(* Logix 5000 project; controller Modbus_TCP_Client_Example vendor 1 type 14 code 154 rev 32.15; software revision 32.05; part 7 of 10 *)

ADD_ON_INSTRUCTION AMP_SCL_Command_Execute   (* revision 1.0 *)
// Applied Motion - SCL Command Execute AOI
// Help:
// The SCL Command Execute AOI executes selected SCL commands (as listed under “Available SCL Commands” in the Host Command Reference).
VAR_IN_OUT
   Input : DINT[14]; {required}   // Drive Input Assembly
   Output : DINT[16]; {required}   // Drive Output Assembly
        [0]   // Command Word
        [10]   // Data/Register 1
        [11]   // Data/Register 2
        [1]   // Jog Speed (0.25 rev/min)
        [2]   // Jog Acceleration (10 rev/s/s)
        [3]   // Jog Deceleration (10 rev/s/s)
        [4]   // Point-to-Point Velocity (0.25 rev/min)
        [5]   // Point-to-Point Acceleration (10 rev/s/s)
        [6]   // Point-to-Point Deceleration (10 rev/s/s)
        [7]   // Point-to-Point Distance (Motor steps)
        [9]   // (2x ASCII Letters in 16 lower word)
END_VAR
VAR_INPUT
   RPI : DINT := 100; {visible}   // Drive Connection Request Packet Interval (milliseconds)
   Execute : BOOL; {required}   // Execute the SCL command
   SCL_Command : INT; {required}   // SCL Command Characters (always 2)
   Reg1 : DINT; {required}   // Data / SCL Register 1
   Reg2 : DINT; {required}   // Data / SCL Register 2
END_VAR
VAR_OUTPUT
   Sent : BOOL; {access Read Only, visible}   // Command has been sent to drive
   In_Progress : BOOL; {access Read Only, visible}   // In progress = sending command
   Done : BOOL; {access Read Only, visible}   // Command sent
   Error : BOOL; {access Read Only, visible}   // Command failed to be sent
   State : DINT := 10; {access Read Only}   // Internal state of progress
END_VAR
VAR
   Loc_StatusCode : AMP_Status_Word;
   Loc_CommandOff_Timer : TIMER;   // Timer to make sure command value was 0 before sending a new command
   Loc_CommandOn_Timer : TIMER;   // Timer to make sure command value is set long enough to be sent to drive
   Loc_Input_Assembly : AMP_Input_Assembly_v2; {access None}
   Loc_Start_ONS : BOOL; {access None}
END_VAR

ROUTINE Logic   (* ladder *)
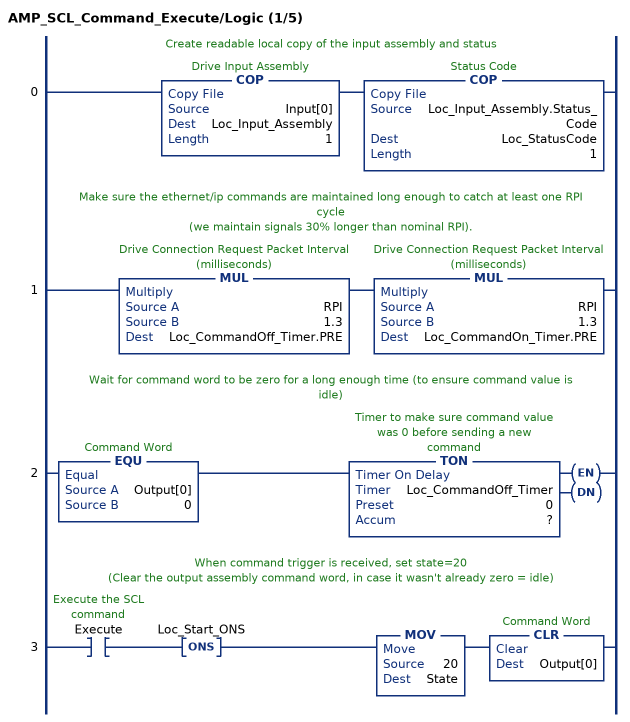
   // Create readable local copy of the input assembly and status
   0: COP(Input[0],Loc_Input_Assembly,1)COP(Loc_Input_Assembly.Status_Code,Loc_StatusCode,1);
   // Make sure the ethernet/ip commands are maintained long enough to catch at least one RPI cycle
   // (we maintain signals 30% longer than nominal RPI).
   1: MUL(RPI,1.3,Loc_CommandOff_Timer.PRE)MUL(RPI,1.3,Loc_CommandOn_Timer.PRE);
   // Wait for command word to be zero for a long enough time (to ensure command value is idle)
   2: EQU(Output[0],0)TON(Loc_CommandOff_Timer,?,?);
   // When command trigger is received, set state=20
   // (Clear the output assembly command word, in case it wasn't already zero = idle)
   3: XIC(Execute)ONS(Loc_Start_ONS)MOV(20,State)CLR(Output[0]);
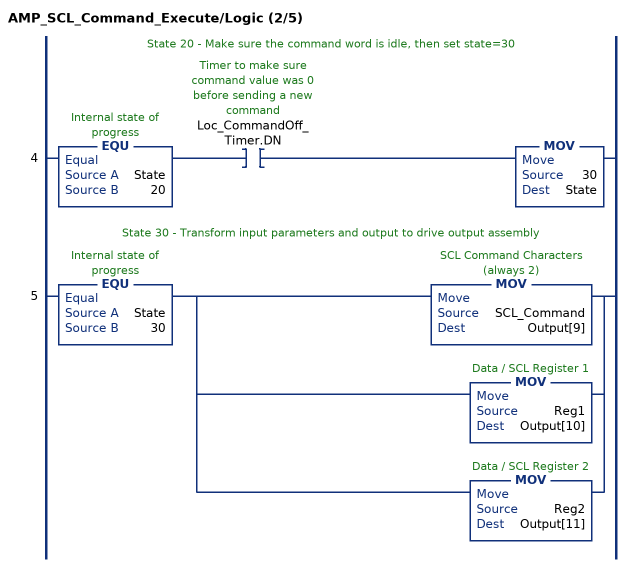
   // State 20 - Make sure the command word is idle, then set state=30
   4: EQU(State,20)XIC(Loc_CommandOff_Timer.DN)MOV(30,State);
   // State 30 - Transform input parameters and output to drive output assembly
   5: EQU(State,30)[MOV(SCL_Command,Output[9]) ,MOV(Reg1,Output[10]) ,MOV(Reg2,Output[11]) ];
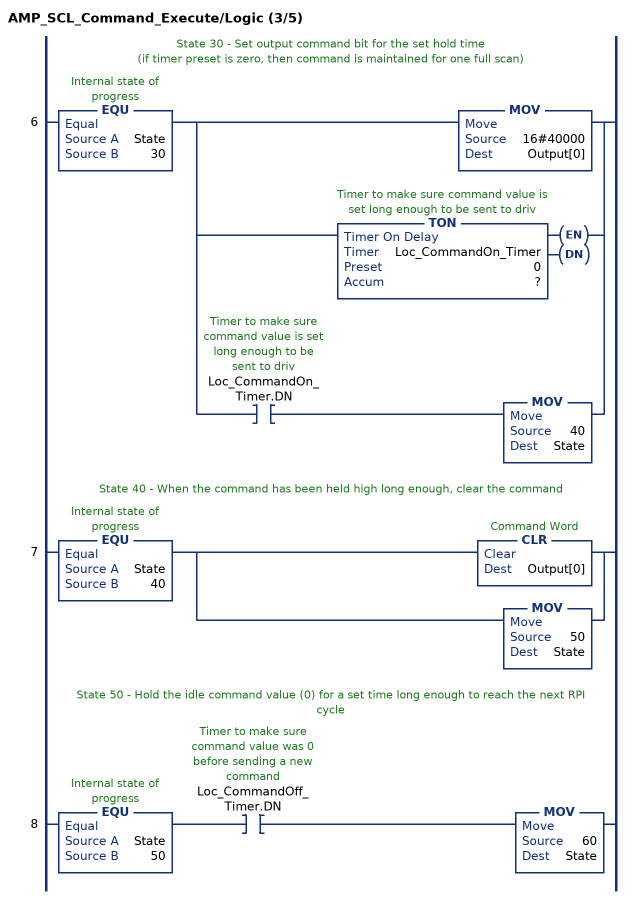
   // State 30 - Set output command bit for the set hold time
   // (if timer preset is zero, then command is maintained for one full scan)
   6: EQU(State,30)[MOV(16#40000,Output[0]) ,TON(Loc_CommandOn_Timer,?,?) ,XIC(Loc_CommandOn_Timer.DN) MOV(40,State) ];
   // State 40 - When the command has been held high long enough, clear the command
   7: EQU(State,40)[CLR(Output[0]) ,MOV(50,State) ];
   // State 50 - Hold the idle command value (0) for a set time long enough to reach the next RPI cycle
   8: EQU(State,50)XIC(Loc_CommandOff_Timer.DN)MOV(60,State);
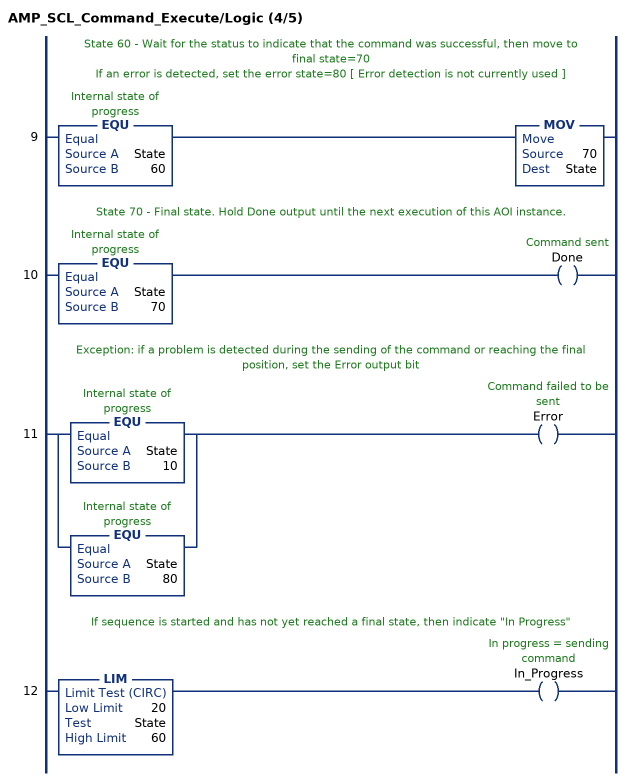
   // State 60 - Wait for the status to indicate that the command was successful, then move to final state=70
   // If an error is detected, set the error state=80 [ Error detection is not currently used ]
   9: EQU(State,60)MOV(70,State);
   // State 70 - Final state. Hold Done output until the next execution of this AOI instance.
   10: EQU(State,70)OTE(Done);
   // Exception: if a problem is detected during the sending of the command or reaching the final position, set the Error output bit
   11: [EQU(State,10) ,EQU(State,80) ]OTE(Error);
   // If sequence is started and has not yet reached a final state, then indicate "In Progress"
   12: LIM(20,State,60)OTE(In_Progress);
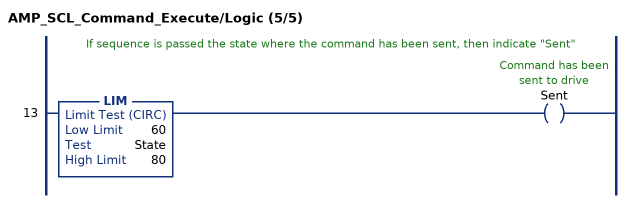
   // If sequence is passed the state where the command has been sent, then indicate "Sent"
   13: LIM(60,State,80)OTE(Sent);
END_ROUTINE
END_ADD_ON_INSTRUCTION

ADD_ON_INSTRUCTION AMP_SCL_Command_Servo   (* revision 1.0, vendor Applied Motion Products Inc. *)
// Applied Motion - Motor SCL Command - AOI
// Help:
// The SCL Command Execute AOI executes selected SCL commands (as listed under “Available SCL Commands” in the reference manual).
VAR_IN_OUT
   Input : DINT[20]; {required}   // Drive Input Assembly
        [4]   // Alarm_Code
        [16]   // Analog_Input1
        [0]   // Control_Word_Received
        [10]   // Position_Error
        [11]   // Actual_Velocity_RPS
        [12]   // Digital_Outputs
        [13]   // Digital_Inputs
        [14]   // Analog_Output1
        [15]   // Analog_Output2
        [17]   // Analog_Input2
        [18]   // Torque_Limit
        [19]   // Second_Encoder_Speed
        [1]   // OpCode1_Received
        [2]   // Control_Mode
        [3]   // Status_Code
        [5]   // Supply_Voltage
        [6]   // Applied_Torque
        [7]   // Drive_Temperature
        [8]   // Encoder_Position
        [9]   // Second_Encoder_Position
   Output : DINT[11]; {required}   // Drive Output Assembly
        [10]   // Reserved
        [4]   // Target Velocity
        [0]   // Control Word
        [3]   // Target Pos
        [1]   // OpCode 1
        [2]   // OpCode 2
        [5]   // Porifle Acceleration
        [6]   // Profile Deceleration
        [7]   // Target Torque
        [8]   // OpCode 3
        [9]   // OpCode 4
END_VAR
VAR_INPUT
   Execute : BOOL; {required}   // Execute the SCL command
   SCL_Command : INT; {required}   // SCL Command Characters (always 2)
   Reg1 : DINT; {required}   // Data / SCL Register 1
   Reg2 : DINT; {required}   // Data / SCL Register 2
END_VAR
VAR_OUTPUT
   Sent : BOOL; {access Read Only, visible}   // Command has been sent to drive
   In_Progress : BOOL; {access Read Only, visible}   // Command in progress
   Done : BOOL; {access Read Only, visible}   // Command completed without errors
   Error : BOOL; {access Read Only, visible}   // Command failed
   State : DINT := 10; {access Read Only}   // Internal state of progress
END_VAR
VAR
   Loc_StatusCode : AMP_Status_Word_Servo; {access None}
   Loc_SCL_ONS : BOOL;
   Loc_Input_Assembly : AMP_Input_Assembly_Servo_v2; {access None}
END_VAR

ROUTINE Logic   (* ladder *)
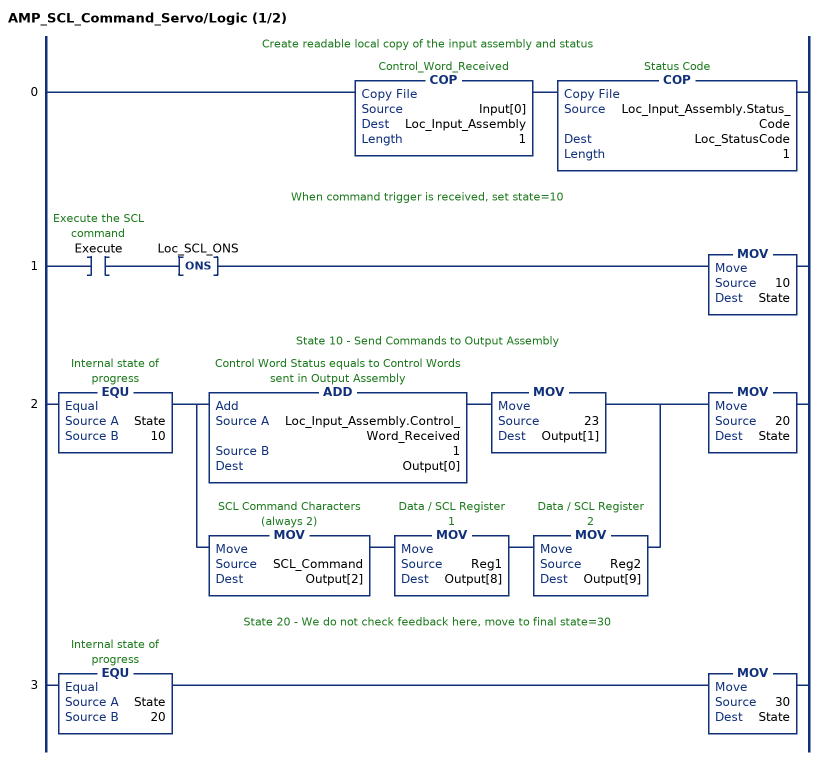
   // Create readable local copy of the input assembly and status
   0: COP(Input[0],Loc_Input_Assembly,1)COP(Loc_Input_Assembly.Status_Code,Loc_StatusCode,1);
   // When command trigger is received, set state=10
   1: XIC(Execute)ONS(Loc_SCL_ONS)MOV(10,State);
   // State 10 - Send Commands to Output Assembly
   2: EQU(State,10)[ADD(Loc_Input_Assembly.Control_Word_Received,1,Output[0]) MOV(23,Output[1]) ,MOV(SCL_Command,Output[2]) MOV(Reg1,Output[8]) MOV(Reg2,Output[9]) ]MOV(20,State);
   // State 20 - We do not check feedback here, move to final state=30
   3: EQU(State,20)MOV(30,State);
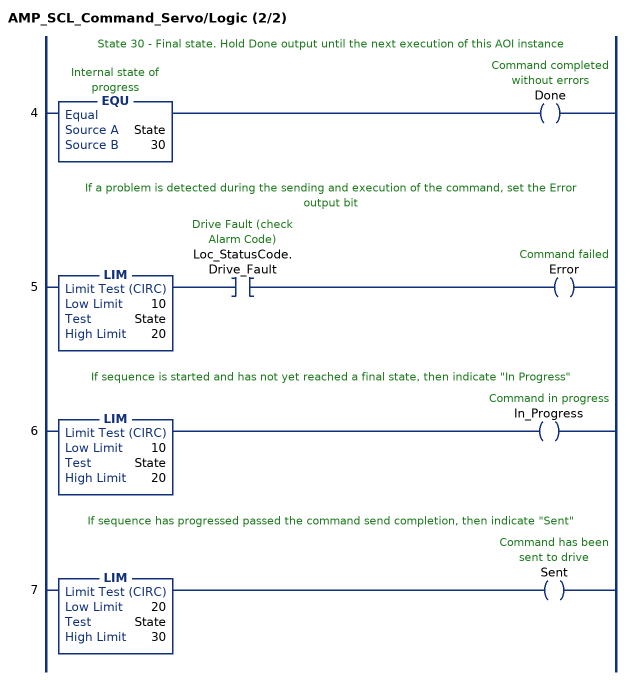
   // State 30 - Final state. Hold Done output until the next execution of this AOI instance
   4: EQU(State,30)OTE(Done);
   // If a problem is detected during the sending and execution of the command, set the Error output bit
   5: LIM(10,State,20)XIC(Loc_StatusCode.Drive_Fault)OTE(Error);
   // If sequence is started and has not yet reached a final state, then indicate "In Progress"
   6: LIM(10,State,20)OTE(In_Progress);
   // If sequence has progressed passed the command send completion, then indicate "Sent"
   7: LIM(20,State,30)OTE(Sent);
END_ROUTINE
END_ADD_ON_INSTRUCTION

ADD_ON_INSTRUCTION AMP_Set_Position_Servo   (* revision 1.0 *)
// Applied Motion - Motor Set Position - AOI
// Help:
// The Motor Enable AOI restores drive current to motor.
VAR_IN_OUT
   Input : DINT[20]; {required}   // Drive Input Assembly
        [4]   // Alarm_Code
        [16]   // Analog_Input1
        [0]   // Control_Word_Received
        [10]   // Position_Error
        [11]   // Actual_Velocity_RPS
        [12]   // Digital_Outputs
        [13]   // Digital_Inputs
        [14]   // Analog_Output1
        [15]   // Analog_Output2
        [17]   // Analog_Input2
        [18]   // Torque_Limit
        [19]   // Second_Encoder_Speed
        [1]   // OpCode1_Received
        [2]   // Control_Mode
        [3]   // Status_Code
        [5]   // Supply_Voltage
        [6]   // Applied_Torque
        [7]   // Drive_Temperature
        [8]   // Encoder_Position
        [9]   // Second_Encoder_Position
   Output : DINT[11]; {required}   // Drive Output Assembly
        [10]   // Reserved
        [4]   // Target Velocity
        [0]   // Control Word
        [3]   // Target Pos
        [1]   // OpCode 1
        [2]   // OpCode 2
        [5]   // Porifle Acceleration
        [6]   // Profile Deceleration
        [7]   // Target Torque
        [8]   // OpCode 3
        [9]   // OpCode 4
END_VAR
VAR_INPUT
   Execute : BOOL; {required}   // Execute the SCL command EP
   Position : DINT; {required}   // Position SetPoint DINT value
END_VAR
VAR_OUTPUT
   Sent : BOOL; {access Read Only, visible}   // Command has been sent to drive
   In_Progress : BOOL; {access Read Only, visible}   // Command in progress
   Done : BOOL; {access Read Only, visible}   // Command completed without errors - Drive is Homed
   Error : BOOL; {access Read Only, visible}   // Command failed
   State : DINT := 10; {access Read Only}   // Internal state of progress
END_VAR
VAR
   Loc_StatusCode : AMP_Status_Word_Servo;
   Loc_Input_Assembly : AMP_Input_Assembly_Servo_v2;
   Loc_SCL_ONS : BOOL;
   Loc_Reg2 : DINT;   // Data / SCL Register 2
   Loc_Reg1 : DINT;   // Data / SCL Register 1
   Loc_SCL_Command : INT := 'EP';   // SCL Command Characters (always 2)
END_VAR

ROUTINE Logic   (* ladder *)
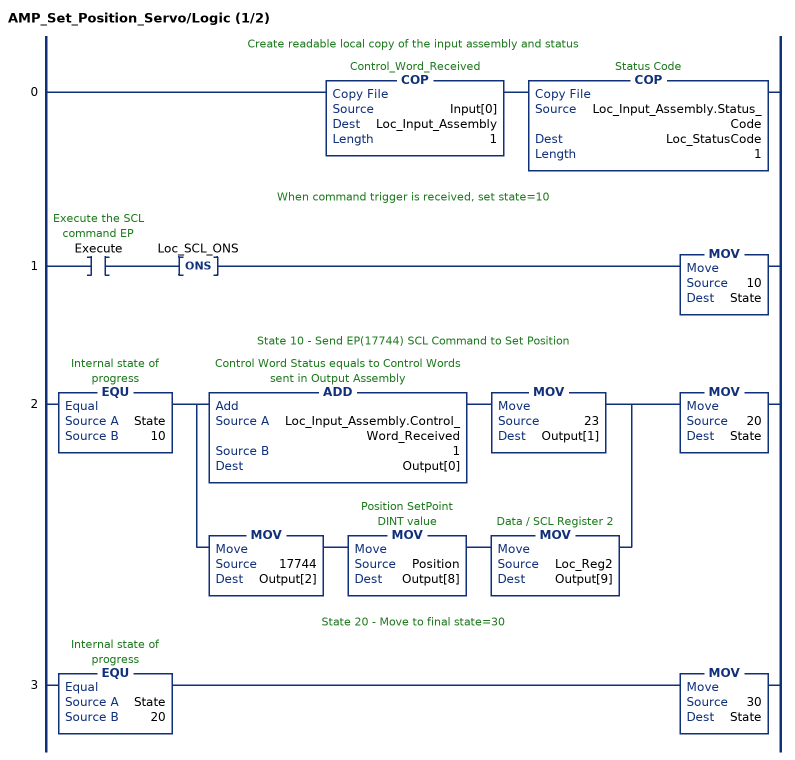
   // Create readable local copy of the input assembly and status
   0: COP(Input[0],Loc_Input_Assembly,1)COP(Loc_Input_Assembly.Status_Code,Loc_StatusCode,1);
   // When command trigger is received, set state=10
   1: XIC(Execute)ONS(Loc_SCL_ONS)MOV(10,State);
   // State 10 - Send EP(17744) SCL Command to Set Position
   2: EQU(State,10)[ADD(Loc_Input_Assembly.Control_Word_Received,1,Output[0]) MOV(23,Output[1]) ,MOV(17744,Output[2]) MOV(Position,Output[8]) MOV(Loc_Reg2,Output[9]) ]MOV(20,State);
   // State 20 - Move to final state=30
   3: EQU(State,20)MOV(30,State);
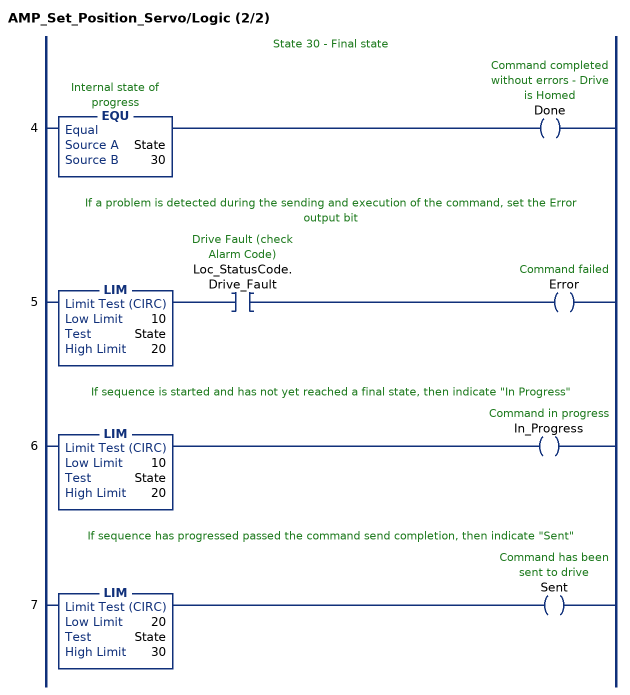
   // State 30 - Final state
   4: EQU(State,30)OTE(Done);
   // If a problem is detected during the sending and execution of the command, set the Error output bit
   5: LIM(10,State,20)XIC(Loc_StatusCode.Drive_Fault)OTE(Error);
   // If sequence is started and has not yet reached a final state, then indicate "In Progress"
   6: LIM(10,State,20)OTE(In_Progress);
   // If sequence has progressed passed the command send completion, then indicate "Sent"
   7: LIM(20,State,30)OTE(Sent);
END_ROUTINE
END_ADD_ON_INSTRUCTION

ADD_ON_INSTRUCTION AMP_Status_Code   (* revision 1.0 *)
// Applied Motion - Status Code AOI
// Help:
// The Status Code AOI uses the raw data stored in the Status Code word (Element 0 from Input Assembly 0x65) to set individual appropriately named boolean outputs.
VAR_INPUT
   Input : DINT; {required}   // Element 0 from Drive Input Assembly (0x65)
END_VAR
VAR_OUTPUT
   Motor_Enabled : BOOL; {access Read Only, visible}
   Sampling : BOOL; {access Read Only, visible}
   Drive_Fault : BOOL; {access Read Only, visible}
   In_Position : BOOL; {access Read Only, visible}
   Moving : BOOL; {access Read Only, visible}
   Jogging : BOOL; {access Read Only, visible}
   Stopping : BOOL; {access Read Only, visible}
   Waiting : BOOL; {access Read Only, visible}
   Saving : BOOL; {access Read Only, visible}
   Alarm_Present : BOOL; {access Read Only, visible}
   Homing : BOOL; {access Read Only, visible}
   Wait_Time : BOOL; {access Read Only, visible}
   Wizard_Running : BOOL; {access Read Only, visible}
   Checking_Encoder : BOOL; {access Read Only, visible}
   Q_Program_Running : BOOL; {access Read Only, visible}
   Initializing : BOOL; {access Read Only, visible}
END_VAR

ROUTINE Logic   (* ladder *)
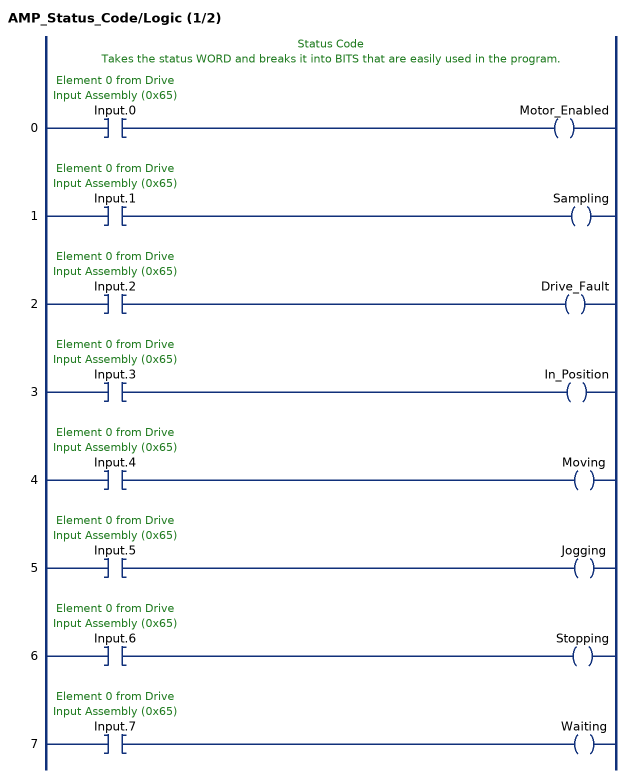
   // Status Code
   // Takes the status WORD and breaks it into BITS that are easily used in the program.
   0: XIC(Input.0)OTE(Motor_Enabled);
   1: XIC(Input.1)OTE(Sampling);
   2: XIC(Input.2)OTE(Drive_Fault);
   3: XIC(Input.3)OTE(In_Position);
   4: XIC(Input.4)OTE(Moving);
   5: XIC(Input.5)OTE(Jogging);
   6: XIC(Input.6)OTE(Stopping);
   7: XIC(Input.7)OTE(Waiting);
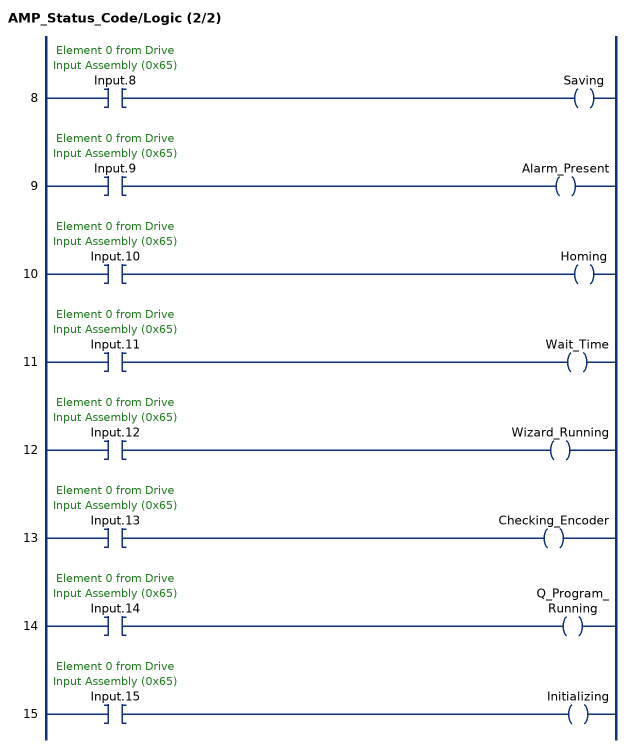
   8: XIC(Input.8)OTE(Saving);
   9: XIC(Input.9)OTE(Alarm_Present);
   10: XIC(Input.10)OTE(Homing);
   11: XIC(Input.11)OTE(Wait_Time);
   12: XIC(Input.12)OTE(Wizard_Running);
   13: XIC(Input.13)OTE(Checking_Encoder);
   14: XIC(Input.14)OTE(Q_Program_Running);
   15: XIC(Input.15)OTE(Initializing);
END_ROUTINE
END_ADD_ON_INSTRUCTION

ADD_ON_INSTRUCTION AMP_Status_Code_Servo   (* revision 1.0, vendor Applied Motion Products Inc. *)
// Applied Motion - Status Code(SC) AOI
// Help:
// The Status Code AOI uses the raw data stored in the Status Code word (Element 0 from Input Assembly) to set individual appropriately named boolean outputs.
VAR_INPUT
   Input : DINT; {required}   // Element 4 from Drive Input Assembly
END_VAR
VAR_OUTPUT
   Motor_Enabled : BOOL; {access Read Only, visible}   // Motor is Enabled(Brake is released if applicable)
   Sampling : BOOL; {access Read Only, visible}   // Sampling (Luna software oscilloscope function opens)
   Drive_Fault : BOOL; {access Read Only, visible}   // Drive has fault, Motor Disabled
   In_Position : BOOL; {access Read Only, visible}   // Motor is in Position, it is standstill
   Moving : BOOL; {access Read Only, visible}   // Motor is Moving
   Jogging : BOOL; {access Read Only, visible}   // Motor is Jogging
   Stopping : BOOL; {access Read Only, visible}   // Motor is Stopping (Decelerating)
   Waiting : BOOL; {access Read Only, visible}   // Wait for Input Signal (e.g. follow WI command)
   Saving : BOOL; {access Read Only, visible}   // Drive is Saving Parameters
   Alarm_Present : BOOL; {access Read Only, visible}   // Dirve has alram present, fault and warning
   Homing : BOOL; {access Read Only, visible}   // Motor is Homing
   Wait_Time : BOOL; {access Read Only, visible}   // Waiting for an input (executing WD or WT command/delay after homing)
   Wizard_Running : BOOL; {access Read Only, visible}   // Wizard Running, Drive internal status
   Checking_Encoder : BOOL; {access Read Only, visible}   // Drive is checking encoder, Drive internal status
   Q_Program_Running : BOOL; {access Read Only, visible}   // Q Program is executing
   Servo_Ready : BOOL; {access Read Only, visible}   // Servo is ready
   CSP_Following : BOOL; {access Read Only, visible}   // CSP following internal status
   In_Velocity : BOOL; {access Read Only, visible}   // Motor is in Velocity
   Zero_Speed : BOOL; {access Read Only, visible}   // Motor is not moving
   Torque_Reached : BOOL; {access Read Only, visible}   // Torque Arrival
   In_Torque : BOOL; {access Read Only, visible}   // Consistent Torque
   Group2_PID : BOOL; {access Read Only, visible}   // The second set of gain is in operation
   Secondary_Control_Mode : BOOL; {access Read Only, visible}   // The second control mode is in operation
   Velocity_Reached : BOOL; {access Read Only, visible}   // Velocity is reached
   Homing_Complete : BOOL; {access Read Only, visible}   // Homing has been completed
END_VAR

ROUTINE Logic   (* ladder *)
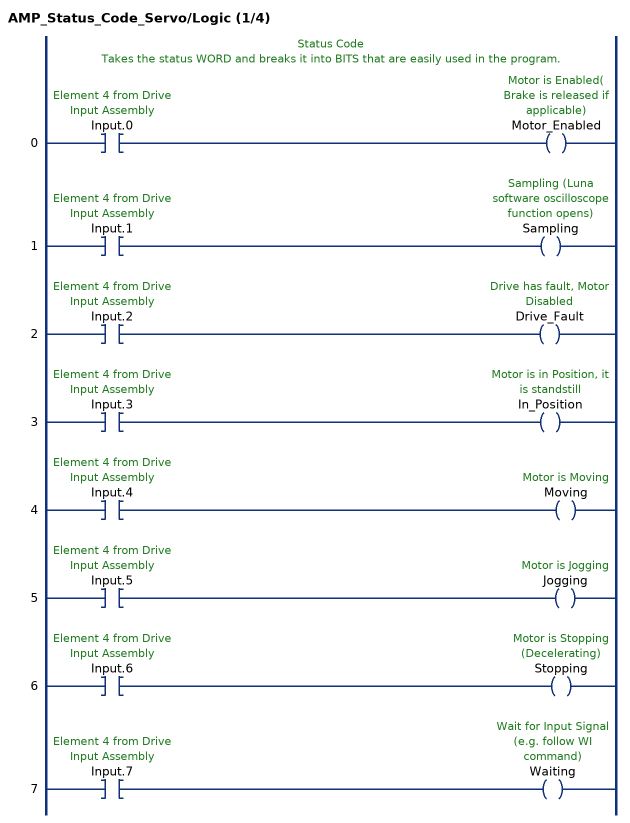
   // Status Code
   // Takes the status WORD and breaks it into BITS that are easily used in the program.
   0: XIC(Input.0)OTE(Motor_Enabled);
   1: XIC(Input.1)OTE(Sampling);
   2: XIC(Input.2)OTE(Drive_Fault);
   3: XIC(Input.3)OTE(In_Position);
   4: XIC(Input.4)OTE(Moving);
   5: XIC(Input.5)OTE(Jogging);
   6: XIC(Input.6)OTE(Stopping);
   7: XIC(Input.7)OTE(Waiting);
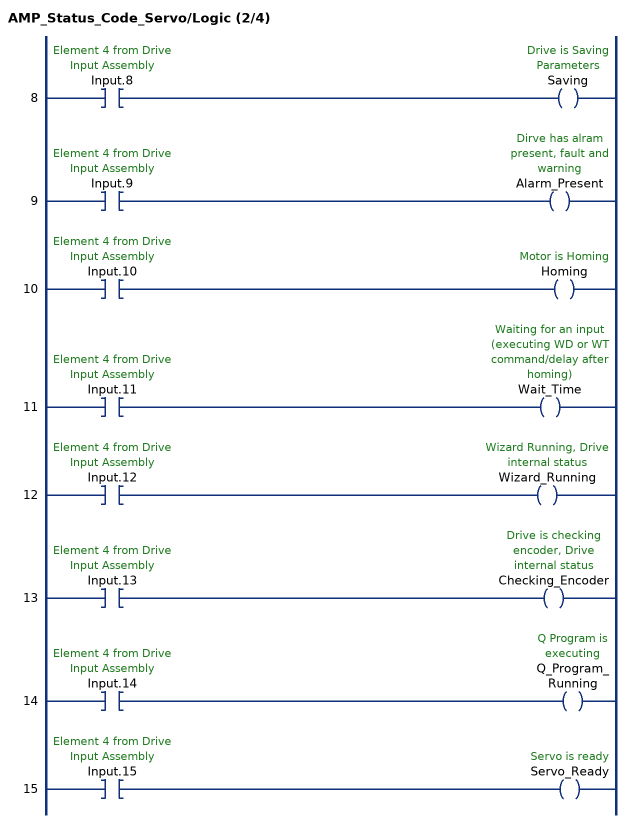
   8: XIC(Input.8)OTE(Saving);
   9: XIC(Input.9)OTE(Alarm_Present);
   10: XIC(Input.10)OTE(Homing);
   11: XIC(Input.11)OTE(Wait_Time);
   12: XIC(Input.12)OTE(Wizard_Running);
   13: XIC(Input.13)OTE(Checking_Encoder);
   14: XIC(Input.14)OTE(Q_Program_Running);
   15: XIC(Input.15)OTE(Servo_Ready);
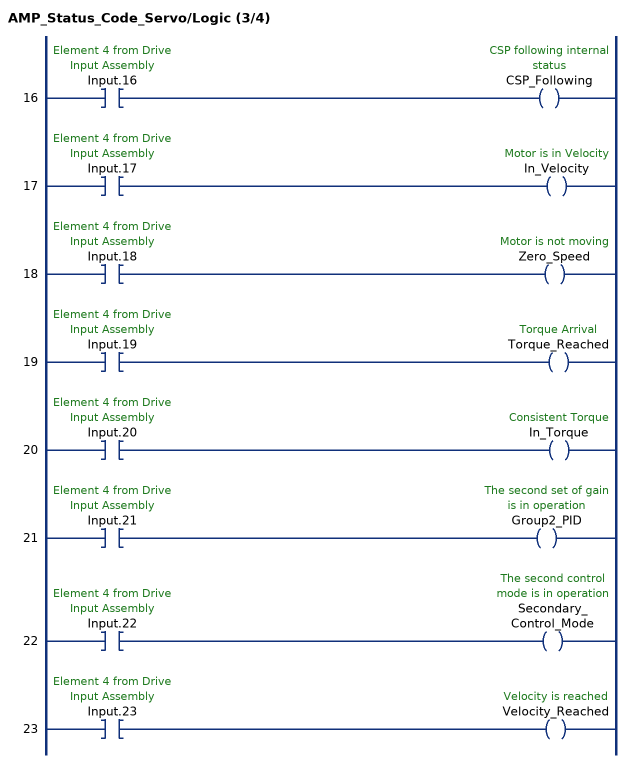
   16: XIC(Input.16)OTE(CSP_Following);
   17: XIC(Input.17)OTE(In_Velocity);
   18: XIC(Input.18)OTE(Zero_Speed);
   19: XIC(Input.19)OTE(Torque_Reached);
   20: XIC(Input.20)OTE(In_Torque);
   21: XIC(Input.21)OTE(Group2_PID);
   22: XIC(Input.22)OTE(Secondary_Control_Mode);
   23: XIC(Input.23)OTE(Velocity_Reached);
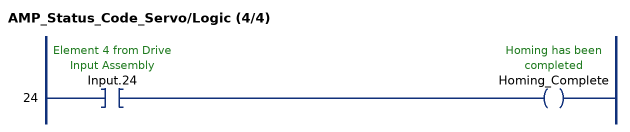
   24: XIC(Input.24)OTE(Homing_Complete);
END_ROUTINE
END_ADD_ON_INSTRUCTION

ADD_ON_INSTRUCTION AMP_Torque_Control_Servo   (* revision 1.0 *)
// Applied Motion - Motor Torque - AOI
// Use Normal/Crash Stop AOI to Stop Torque
// Help:
// The AOI switch Control mode to Torque mode and apply Torque. Use Normal stop or Crash stop AOI to stop applying torque.
// Target Torque Percentage is Limit by Torque Limit shown in Input Assembly.
VAR_IN_OUT
   Input : DINT[20]; {required}   // Drive Input Assembly
        [16]   // Analog_Input1
        [4]   // Alarm_Code
        [0]   // Control_Word_Received
        [10]   // Position_Error
        [11]   // Actual_Velocity_RPS
        [12]   // Digital_Outputs
        [13]   // Digital_Inputs
        [14]   // Analog_Output1
        [15]   // Analog_Output2
        [17]   // Analog_Input2
        [18]   // Torque_Limit
        [19]   // Second_Encoder_Speed
        [1]   // OpCode1_Received
        [2]   // Control_Mode
        [3]   // Status_Code
        [5]   // Supply_Voltage
        [6]   // Applied_Torque
        [7]   // Drive_Temperature
        [8]   // Encoder_Position
        [9]   // Second_Encoder_Position
   Output : DINT[11]; {required}   // Drive Output Assembly
        [10]   // Reserved
        [4]   // Target Velocity
        [0]   // Control Word
        [3]   // Target Pos
        [1]   // OpCode 1
        [2]   // OpCode 2
        [5]   // Porifle Acceleration
        [6]   // Profile Deceleration
        [7]   // Target Torque
        [8]   // OpCode 3
        [9]   // OpCode 4
END_VAR
VAR_INPUT
   Start : BOOL; {required}   // Start Applying Torque (on rising edge)
   Target_Torque_Percentage : INT := 10; {required}   // Target Torque Percentage, for reverse direction use Negative value
   Torque_Ramp : INT; {required}   // Torque Ramp (0.1%/sec)
   Speed_Limit_rps : REAL; {required}   // Torque Speed Limit in rps
   Acc : REAL; {required}   // Acceleration rev/s/s
   Dec : REAL; {required}   // Deceleration rev/s/s
END_VAR
VAR_OUTPUT
   Sent : BOOL; {access Read Only, visible}   // Command has been sent to drive
   In_Progress : BOOL; {access Read Only, visible}   // Command is in progress
   Done : BOOL; {access Read Only, visible}   // Command completed without errors
   Error : BOOL; {access Read Only, visible}   // Command Failed
   State : DINT := 10; {access Read Only}   // Internal state of progress
END_VAR
VAR
   Loc_StatusCode : AMP_Status_Word_Servo;
   Loc_Input_Assembly : AMP_Input_Assembly_Servo_v2;
   Loc_Torque_ONS : BOOL;
   Loc_Command_Wait : TIMER := (PRE := 100); {access None}   // Wait Timer for New Command
END_VAR

ROUTINE Logic   (* ladder *)
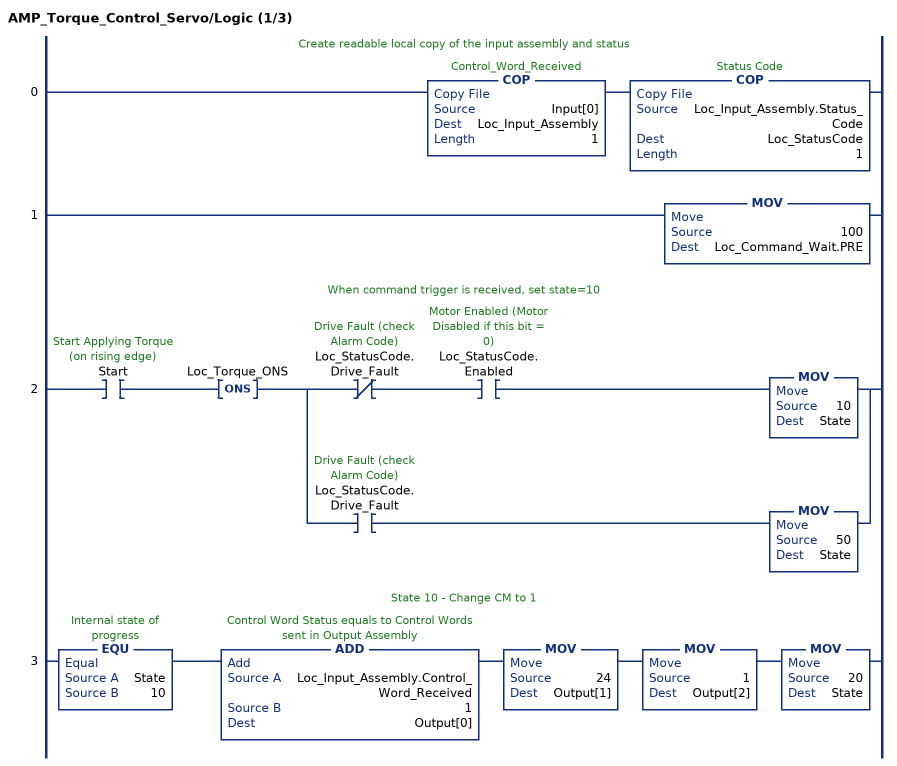
   // Create readable local copy of the input assembly and status
   0: COP(Input[0],Loc_Input_Assembly,1)COP(Loc_Input_Assembly.Status_Code,Loc_StatusCode,1);
   1: MOV(100,Loc_Command_Wait.PRE);
   // When command trigger is received, set state=10
   2: XIC(Start)ONS(Loc_Torque_ONS)[XIO(Loc_StatusCode.Drive_Fault) XIC(Loc_StatusCode.Enabled) MOV(10,State) ,XIC(Loc_StatusCode.Drive_Fault) MOV(50,State) ];
   // State 10 - Change CM to 1
   3: EQU(State,10)ADD(Loc_Input_Assembly.Control_Word_Received,1,Output[0])MOV(24,Output[1])MOV(1,Output[2])MOV(20,State);
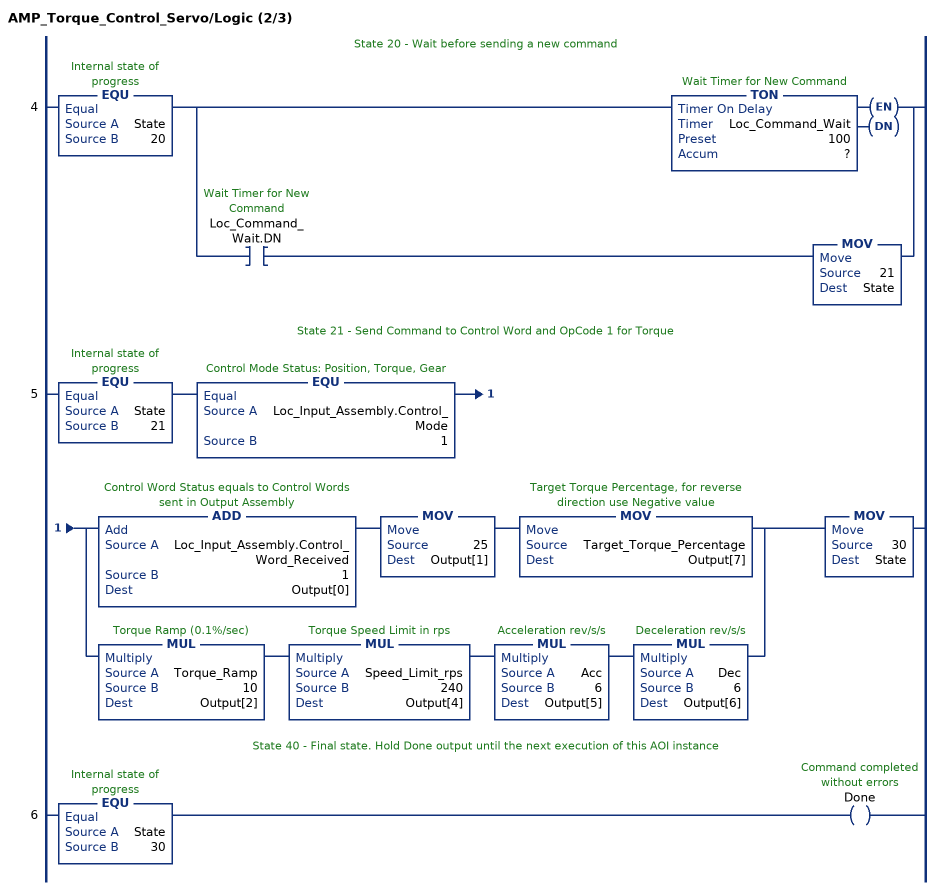
   // State 20 - Wait before sending a new command
   4: EQU(State,20)[TON(Loc_Command_Wait,?,?) ,XIC(Loc_Command_Wait.DN) MOV(21,State) ];
   // State 21 - Send Command to Control Word and OpCode 1 for Torque
   5: EQU(State,21)EQU(Loc_Input_Assembly.Control_Mode,1)[ADD(Loc_Input_Assembly.Control_Word_Received,1,Output[0]) MOV(25,Output[1]) MOV(Target_Torque_Percentage,Output[7]) ,MUL(Torque_Ramp,10,Output[2]) MUL(Speed_Limit_rps,240,Output[4]) MUL(Acc,6,Output[5]) MUL(Dec,6,Output[6]) ]MOV(30,State);
   // State 40 - Final state. Hold Done output until the next execution of this AOI instance
   6: EQU(State,30)OTE(Done);
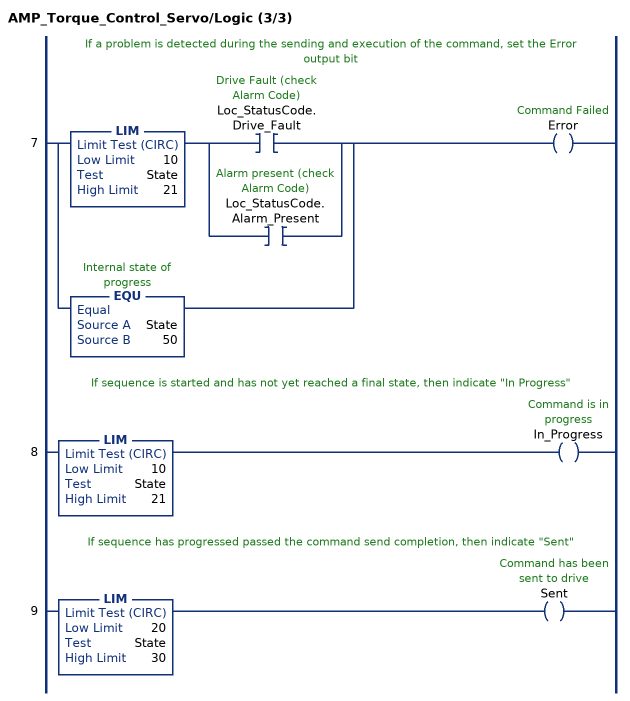
   // If a problem is detected during the sending and execution of the command, set the Error output bit
   7: [LIM(10,State,21) [XIC(Loc_StatusCode.Drive_Fault) ,XIC(Loc_StatusCode.Alarm_Present) ] ,EQU(State,50) ]OTE(Error);
   // If sequence is started and has not yet reached a final state, then indicate "In Progress"
   8: LIM(10,State,21)OTE(In_Progress);
   // If sequence has progressed passed the command send completion, then indicate "Sent"
   9: LIM(20,State,30)OTE(Sent);
END_ROUTINE
END_ADD_ON_INSTRUCTION
